RoboDK station: LEGOS_RDK.rdk

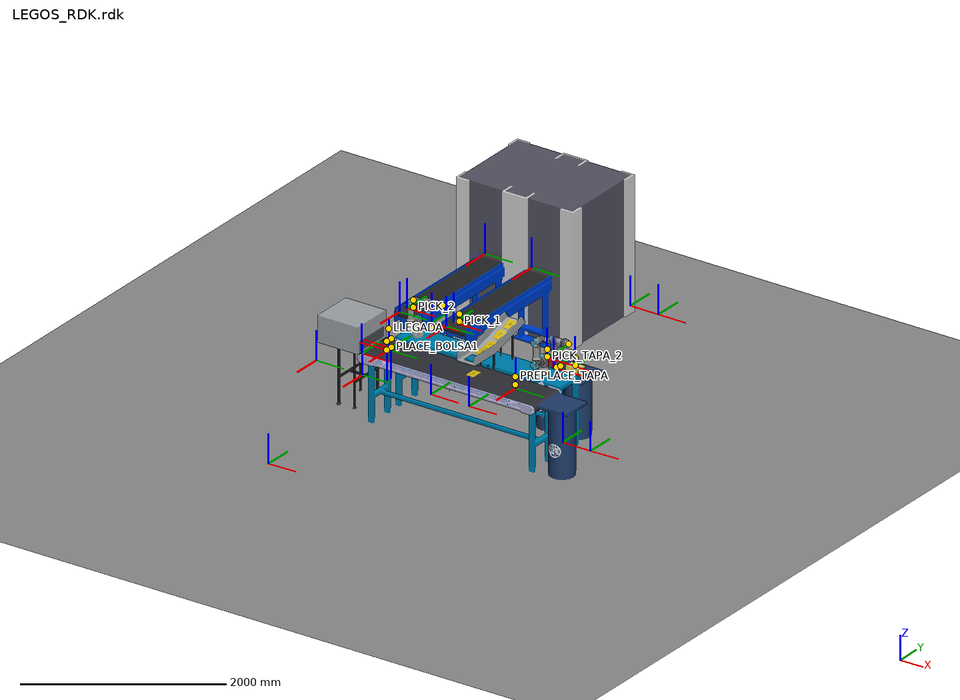
[picture v0: the station drawn from its stored meshes, robots at their saved joint values, targets as dots, program paths as lines]
Station LEGOS_RDK (saved by RoboDK 5.9.4). Poses are relative to the parent item; angles as X-Y-Z fixed-axis rotations.
Station parameters (name, value as stored): SenyalSensor_C, 0, SenyalSensor_T, 0, BOLSA2_PICK, 1, BOLSA1_PICK, 1, Continuar1, 1, PRIMERA_RUN, 1, SenyalSensor_I, 0, TOTAL_PEDIDO_1, 0, TOTAL_PEDIDO_2, 0, ACTIVO, 1, PP_BOLSA_2, 0, INS_BOLSA_2, 0, TAPA_BOLSA_2, 0, Conti_T, 1, lim_ins, 0, lim_tapa, 0, PARAR_ESTACION, 1, CICLOS_HASTA_PARAR, 0, PP_LOCAL, 0, IO_0, 0, Cinta_Terminada, 0, Conti_I, 1, MQTT_ESTACION_ENCENDIDA, 0, PARADA_EMERGENCIA, 0, INITIAL_P1, 0, CONTADOR_C, 2, CONTADOR_T, 2, lim_bolsa, 0, TOTAL_PEDIDO_2_INICIAL, 2, CONTADOR_I, 2, PEDIDO_1_INICIAL, 2, PEDIDO_2_INICIAL, 0, LIMITE_TAPAS, 0, LIMITE_INSTRU, 0, LIMITE_BOLSAS, 0, R1_LIBRE, 1, R2_LIBRE, 1, INSTRU_LIBRE, 1, PRODUCIR_CAJAS, 0, NUMERO_PEDIDO, PED_1779911272, STOCK_VERIFICADO, 1, ES_REANUDACION, 0, CONTADOR_CREADAS, 2, MAPA_CAJA_001, CAJA_001, MAPA_CAJA_002, CAJA_002, MAPA_CAJA_003, CAJA2_003, NOMBRE_C_001, CAJA_001, NOMBRE_C_002, CAJA_002, NOMBRE_T_001, instru_2, NOMBRE_T_002, instru_2, NOMBRE_T_003, instru_2, NOMBRE_C_003, CAJA2_003, NOMBRE_C_004, CAJA_004, MAPA_CAJA_004, CAJA_004, NOMBRE_C_005, CAJA_005, MAPA_CAJA_005, CAJA_005, NOMBRE_C_006, CAJA_005, MAPA_CAJA_006, CAJA_006, NOMBRE_C_007, CAJA_007, NOMBRE_T_004, instru_2, MAPA_CAJA_007, CAJA_007, NOMBRE_C_008, CAJA_008, NOMBRE_T_005, instru_2, MAPA_CAJA_008, CAJA_008, NOMBRE_C_009, CAJA_008, NOMBRE_T_006, instru_2, MAPA_CAJA_009, CAJA_009, NOMBRE_C_010, CAJA_010, NOMBRE_T_007, instru_2, MAPA_CAJA_010, CAJA_010, NOMBRE_T_008, instru_2, NOMBRE_T_009, instru_2, NOMBRE_T_010, instru_2, NOMBRE_CAJA_EN_T
  - frame ROBOT1 at (240, 410, 60) mm
    - frame Frame PEDESTAL (OBJETO 1) at (280, 230, -915) mm
      - frame COGIDA_1 at (-110, -105, 915) mm
        - target PICK_1 (Cartesian target) at (46.65, 33, 11.24) mm, rotated rx 180 ry 0 rz 0 deg; joints [76.028, -114.59, -95.798, -59.613, 90, -13.972] of r_UR3e_(COGIDA)
        - target PREPICK_1 (Cartesian target) at (46.65, 33, 90) mm, rotated rx 180 ry 0 rz 0 deg; joints [76.028, -108.102, -82.469, -79.429, 90, -13.972] of r_UR3e_(COGIDA)
    - frame Frame PEDESTAL (OBJETO 2) at (-170, 230, -915) mm
      - frame COGIDA_2 at (-210, -105, 915) mm
        - target PICK_2 (Cartesian target) at (46.65, 33, 11.24) mm, rotated rx 180 ry 0 rz 0 deg; joints [76.028, -114.59, -95.798, -59.613, 90, -13.972] of r_UR3e_(COGIDA)
        - target PREPICK_2 (Cartesian target) at (46.65, 33, 90) mm, rotated rx 180 ry 0 rz 0 deg; joints [76.028, -108.102, -82.469, -79.429, 90, -13.972] of r_UR3e_(COGIDA)
    - frame CircuitConveyor Base at (80, 125, -65) mm, rotated rx 0 ry 0 rz -90 deg
      - robot CircuitConveyorDoor: 1 axes
          modified DH rows (alpha deg, a mm, theta deg, d mm): 0, 0, 0, 0 linear
          joint limits [0] to [80]; home [0]; saved at [0]
      - frame CircuitConveyorRef_Init at (-1430, 10, 60) mm
        - object BOLSA 1 at (-120, 40, 0) mm, rotated rx 0 ry 0 rz -90 deg, size 93 x 60 x 20.1 mm, geometry from tinker.obj
      - robot CircuitConveyor: 1 axes
          modified DH rows (alpha deg, a mm, theta deg, d mm): 0, 0, 0, 0 linear
          base shift (0, 0, 0) mm, rotated rx 0 ry 90 rz 0 deg
          joint limits [-200000] to [200000]; home [0]; saved at [1430]
        - frame CircuitConveyorRef at (0, 10, 50) mm
          - object BOLSA 1 at (-1550, 40, 10) mm, rotated rx 0 ry 0 rz -90 deg, size 93 x 60 x 20.1 mm, geometry from tinker.obj
    - frame CircuitConveyor Base(2) at (-470, 125, -65) mm, rotated rx 0 ry 0 rz -90 deg
      - robot CircuitConveyorDoor(2): 1 axes
          modified DH rows (alpha deg, a mm, theta deg, d mm): 0, 0, 0, 0 linear
          joint limits [0] to [80]; home [0]; saved at [0]
      - frame CircuitConveyorRef_Init(2) at (-1430, 10, 60) mm
        - object BOLSA 2 at (-120, 40, 0) mm, rotated rx 0 ry 0 rz -90 deg, size 93 x 60 x 20.1 mm, geometry from tinker.obj
      - robot CircuitConveyor(2): 1 axes
          modified DH rows (alpha deg, a mm, theta deg, d mm): 0, 0, 0, 0 linear
          base shift (0, 0, 0) mm, rotated rx 0 ry 90 rz 0 deg
          joint limits [-200000] to [200000]; home [0]; saved at [1430]
        - frame CircuitConveyorRef(2) at (0, 10, 50) mm
          - object BOLSA 2 at (-1550, 40, 10) mm, rotated rx 0 ry 0 rz -90 deg, size 93 x 60 x 20.1 mm, geometry from tinker.obj
  - frame ROBOT 2 at (1680, 410, -20) mm
    - frame Frame PEDESTAL (PACK 2) at (-50, 230, -915) mm
      - object Pedestal H36in (Type 1) at (-110, -60, -69) mm, size 400 x 400 x 914.4 mm, geometry from Pedestal-H36in-Type-1.sld
      - object dispensa_tapas at (-122, -131, 835) mm, size 162 x 117 x 81 mm, geometry from tinker.obj
      - frame COGIDA_TAPA_2 at (-110, -105, 922) mm
        - target PICK_TAPA_2 (Cartesian target) at (0, 0, 11.24) mm, rotated rx 180 ry 0 rz 0 deg; joints [76.028, -114.59, -95.798, -59.613, 90, -13.972] of r_UR3e_(COGIDA)
        - target PREPICK_TAPA_2 (Cartesian target) at (0, 0, 90) mm, rotated rx 180 ry 0 rz 0 deg; joints [76.028, -108.102, -82.469, -79.429, 90, -13.972] of r_UR3e_(COGIDA)
        - frame FrameInitTapa_2 at (0, 1410, 0) mm
          - object TAPA at (-72, -1477.5, -10) mm, rotated rx 0 ry 0 rz 90 deg, size 111 x 156 x 21 mm, geometry from tinker.obj
        - object TAPA at (-72, -67.5, -10) mm, rotated rx 0 ry 0 rz 90 deg, size 111 x 156 x 21 mm, geometry from tinker.obj
    - frame Frame PEDESTAL (PACK 1) at (280, 230, -915) mm
      - object Pedestal H36in (Type 1) at (-110, -60, -69) mm, size 400 x 400 x 914.4 mm, geometry from Pedestal-H36in-Type-1.sld
      - object dispensa_tapas at (-122, -131, 835) mm, size 162 x 117 x 81 mm, geometry from tinker.obj
      - frame COGIDA_TAPA at (-110, -105, 922) mm
        - target PICK_TAPA (Cartesian target) at (0, 0, 11.24) mm, rotated rx 180 ry 0 rz 0 deg; joints [76.028, -114.59, -95.798, -59.613, 90, -13.972] of r_UR3e_(COGIDA)
        - target PREPICK_TAPA (Cartesian target) at (0, 0, 90) mm, rotated rx 180 ry 0 rz 0 deg; joints [76.028, -108.102, -82.469, -79.429, 90, -13.972] of r_UR3e_(COGIDA)
        - frame FrameInitTapa at (0, 1410, 0) mm
          - object TAPA at (-72, -1477.5, -10) mm, rotated rx 0 ry 0 rz 90 deg, size 111 x 156 x 21 mm, geometry from tinker.obj
        - object TAPA at (-72, -67.5, -10) mm, rotated rx 0 ry 0 rz 90 deg, size 111 x 156 x 21 mm, geometry from tinker.obj
  - frame FrameCintaP at (0, -440, 0) mm
    - robot CINTA_PRINCIPAL: 1 axes
        modified DH rows (alpha deg, a mm, theta deg, d mm): 0, 0, 0, 0 linear
        base shift (0, 0, 0) mm, rotated rx 0 ry 90 rz 0 deg
        joint limits [-500000] to [500000]; home [0]; saved at [0]
      - frame FrameCAJA at (170, 220, 0) mm, rotated rx 0 ry 0 rz -90 deg
    - object MesaCinta at (1040, 170, -770) mm, rotated rx 0 ry 0 rz -90 deg, size 320 x 2000 x 740 mm, geometry from tinker.obj
    - object Fotocelula_T at (1688, 448, 0) mm, rotated rx 90 ry 0 rz -90 deg, size 683.3 x 45.2 x 12.5 mm, geometry from SICK-WL4S-Laser-Sensor.sld
    - object Fotocelula_C at (188, 448, 0) mm, rotated rx 90 ry 0 rz -90 deg, size 683.3 x 45.2 x 12.5 mm, geometry from SICK-WL4S-Laser-Sensor.sld
    - object Fotocelula_I at (1188, 448, 0) mm, rotated rx 90 ry 0 rz -90 deg, size 683.3 x 45.2 x 12.5 mm, geometry from SICK-WL4S-Laser-Sensor.sld
    - frame COGIDA CINTA at (170, 220, 0) mm, rotated rx 0 ry 0 rz -90 deg
      - target LLEGADA (Cartesian target) at (0.04, 0.12, 230.39) mm, rotated rx -180 ry 0 rz -90 deg; joints [-75.94, -132.382, -21.795, -115.824, 90, 14.06] of r_UR3e_(COGIDA)
      - frame DEJAR_BOLSA1 at (-35, 2, 5) mm, rotated rx -180 ry 0 rz -90 deg
        - target PREPLACE_BOLSA1 (Cartesian target) at (0, 0, -100) mm; joints [-74.482, -118.64, -79.498, -71.862, 90, -344.482] of r_UR3e_(COGIDA)
        - target PLACE_BOLSA1 (Cartesian target) at (0, 0, -8) mm; joints [-74.482, -129.029, -89.848, -51.123, 90, -344.482] of r_UR3e_(COGIDA)
      - frame DEJAR_BOLSA2 at (35, 2, 5) mm, rotated rx -180 ry 0 rz -90 deg
        - target PREPLACE_BOLSA2 (Cartesian target) at (0, 0, -100) mm; joints [-74.482, -118.64, -79.498, -71.862, 90, -344.482] of r_UR3e_(COGIDA)
        - target PLACE_BOLSA2 (Cartesian target) at (0, 0, -8) mm; joints [-74.482, -129.029, -89.848, -51.123, 90, -344.482] of r_UR3e_(COGIDA)
    - frame LLEGADA CINTA at (1670, 220, 0) mm, rotated rx 0 ry 0 rz -90 deg
      - target PREPLACE_TAPA (Cartesian target) at (0, 0, 130) mm, rotated rx 180 ry 0 rz 180 deg; joints [-73.448, -126.178, -60.342, -83.48, 90, 106.552] of r_UR3e_(TAPAS)
      - target PLACE_TAPA (Cartesian target) at (0, 0, 45) mm, rotated rx 180 ry 0 rz 180 deg; joints [-73.448, -132.236, -73.608, -64.156, 90, 106.552] of r_UR3e_(TAPAS)
    - frame Frame_Mec_Cai at (-312, -1127, -825) mm
      - robot Mecanismo_Caida: 1 axes
          modified DH rows (alpha deg, a mm, theta deg, d mm): 0, 0, 0, 0 linear
          base shift (0, 0, 0) mm, rotated rx 0 ry 0 rz 90 deg
          joint limits [-163] to [0]; home [0]; saved at [-163]
    - frame Frame_dis_ins at (1170, 220, 0) mm, rotated rx 0 ry 0 rz -90 deg
      - object Dispensa_instru at (-180, 320, -270) mm, rotated rx 0 ry 0 rz 90 deg, size 216 x 857.7 x 462.8 mm, geometry from tinker.obj
      - object instru2 at (-20, -15, 180) mm, size 126 x 90 x 9.1 mm, geometry from tinker.obj
      - object Square at (0, 0, -10) mm, size 75 x 75 x 0 mm, geometry from Square.sld
    - frame FrameInitInstru at (0, 1410, 0) mm
      - object instru at (1155, -1170, 20) mm, rotated rx 0 ry 0 rz -90 deg, size 126 x 90 x 9.1 mm, geometry from tinker.obj
      - object instru_2 at (1155, -1170, 20) mm, rotated rx 0 ry 0 rz -90 deg, size 126 x 90 x 9.1 mm, geometry from tinker.obj
    - frame FrameInitCaja at (-330, 220, 0) mm, rotated rx 0 ry 0 rz -90 deg
      - object CAJA_REF at (-33, 18, 0) mm, size 105 x 150 x 39 mm, geometry from tinker.obj
      - object CAJA_REF_2 at (-33, 18, 0) mm, size 105 x 150 x 39 mm, geometry from tinker.obj
    - frame Frame_Disp_caj at (-312, 253, -825) mm
      - robot Dispensa_CAJAS: 1 axes
          modified DH rows (alpha deg, a mm, theta deg, d mm): 0, 0, 0, 0 linear
          base shift (0, 0, 0) mm, rotated rx 0 ry 0 rz 90 deg
          joint limits [0] to [120]; home [0]; saved at [0]
    - frame Frame_Caja_completa at (2330, 190, -850) mm, rotated rx 0 ry 0 rz 180 deg
      - object Pedestal H36in (Type 1) at (100, -20, -65) mm, size 400 x 400 x 914.4 mm, geometry from Pedestal-H36in-Type-1.sld
  - folder ROBOTS
    - frame UR3e_Base at (190, 240, -20) mm
      - robot r_UR3e_(COGIDA) (model UR3e): 6 axes, payload 3 kg, reach 500 mm, repeatability 0.03 mm, weight 11 kg
          modified DH rows (alpha deg, a mm, theta deg, d mm): 0, 0, 0, 151.9; 90, 0, 180, 0; 0, 243.55, 0, 0; 0, 213.2, 0, 131.05; -90, 0, 0, 85.35; 90, 0, 180, 92.1
          joint limits [-360, -360, -360, -360, -360, -360] to [360, 360, 360, 360, 360, 360]; home [0, -90, -90, 0, 90, 0]; saved at [0, -90, -90, 0, 90, 0]
        - tool VENTOSA-COG, TCP at (0, 0, 82.18) mm, size 70 x 70 x 80.4 mm
      - target HOME_R1 (Cartesian target) at (387.48, -131.05, 480.8) mm, rotated rx -90 ry 0 rz -90 deg; joints [37.926, -98.256, -58.971, -22.773, 52.074, 0] of r_UR3e_(COGIDA)
      - target SAFE_R1 (Cartesian target) at (298.55, -131.05, 221.17) mm, rotated rx -180 ry 0 rz -90 deg; joints [28.318, -100.412, -56.382, -113.206, 90, 28.318] of r_UR3e_(COGIDA)
      - target PUNTO_PASO_R1 (Cartesian target) at (319.11, -229.65, 250.13) mm, rotated rx -179.97 ry -0.01 rz -92.3 deg; joints [-16.27, -108.19, -60.7, -101.08, 90, -13.97] of r_UR3e_(COGIDA)
    - frame UR3e Base (2) at (1680, 240, -20) mm
      - robot r_UR3e_(TAPAS) (model UR3e): 6 axes, payload 3 kg, reach 500 mm, repeatability 0.03 mm, weight 11 kg
          modified DH rows (alpha deg, a mm, theta deg, d mm): 0, 0, 0, 151.9; 90, 0, 180, 0; 0, 243.55, 0, 0; 0, 213.2, 0, 131.05; -90, 0, 0, 85.35; 90, 0, 180, 92.1
          joint limits [-360, -360, -360, -360, -360, -360] to [360, 360, 360, 360, 360, 360]; home [0, -90, -90, 0, 90, 0]; saved at [0, -90, -90, 0, 90, 0]
        - tool VENTOSA-FIN, TCP at (0, 0, 82.18) mm, size 70 x 70 x 80.4 mm
      - target HOME_R2 (Cartesian target) at (387.48, -131.05, 480.8) mm, rotated rx -90 ry 0 rz -90 deg; joints [37.926, -98.256, -58.971, -22.773, 52.074, 0] of r_UR3e_(COGIDA)
      - target SAFE_R2 (Cartesian target) at (298.55, -131.05, 221.17) mm, rotated rx -180 ry 0 rz -90 deg; joints [28.318, -100.412, -56.382, -113.206, 90, 28.318] of r_UR3e_(COGIDA)
      - target PUNTO_PASO_R2 (Cartesian target) at (319.11, -229.65, 250.13) mm, rotated rx -179.97 ry -0.01 rz -92.3 deg; joints [-16.27, -108.19, -60.7, -101.08, 90, -13.97] of r_UR3e_(COGIDA)
      - target Target 4 (Cartesian target) at (298.55, -131.05, 221.17) mm, rotated rx -180 ry 0 rz -90 deg; joints [0, -90, -90, -90, 90, 0] of r_UR3e_(TAPAS)
  - folder OBJETOS SUELTOS
    - object Floor at (860, -90, -760) mm, size 9000 x 9000 x 0 mm, geometry from Floor.sld
    - frame Frame MESA_ROBOT at (940, 230, 0) mm
      - object Mesa_robots at (100, -40, -760) mm, rotated rx 0 ry 0 rz -90 deg, size 320 x 2000 x 740 mm, geometry from tinker.obj
  - folder PROGRAMAS PYTHON
    - Python program DetectaSensor (listed below)
    - Python program DISPENSAR_B1 (listed below)
    - Python program DISPENSAR_B2 (listed below)
    - Python program REPONER_TAPA (listed below)
    - Python program REPONER_TAPA_2 (listed below)
    - Python program PONER_INSTRU (listed below)
  - folder PROGRAMAS ROBOTS
    - Python program ROBOT1_BOLSA1 (listed below)
    - Python program ROBOT1_BOLSA2 (listed below)
    - Python program ROBOT2_TAPA1 (listed below)
    - Python program ROBOT2_TAPA2 (listed below)
  - Python program MAIN_PRODUCCION (listed below)
  - Python program MqttListener (listed below)
  - Python program BASE_DATOS (listed below)

--- Python program DetectaSensor ---
import time
from robodk import robolink
from robodk import robomath

"""
DetectaSensor.py — Script vigía de fotocélulas.
Corre como proceso independiente en paralelo con main_produccion.
Detecta colisiones entre las cajas del FrameCAJA y las tres fotocélulas
(C, I, T) y actualiza los params SenyalSensor_* en RoboDK.
Desde esta versión también escribe el NOMBRE de la caja detectada en
cada sensor ANTES de actualizar la señal, para que Base_datos pueda
identificar unívocamente qué caja física pasó por cada punto.
Se comunica con el resto de scripts ÚNICAMENTE vía RDK.setParam/getParam.
"""

RDK = robolink.Robolink()
RDK.COM.settimeout(10)

REFERENCE_FRAME = 'FrameCAJA'

frame = RDK.Item(REFERENCE_FRAME, robolink.ITEM_TYPE_FRAME)

fotocelulaC = RDK.Item('Fotocelula_C')
fotocelulaT = RDK.Item('Fotocelula_T')
fotocelulaI = RDK.Item('Fotocelula_I')

estado_detectadoC = -1
estado_detectadoT = -1
estado_detectadoI = -1

if not frame.Valid():
    raise Exception(f'El frame "{REFERENCE_FRAME}" no es válido o no existe.')

if not fotocelulaC.Valid() or not fotocelulaT.Valid() or not fotocelulaI.Valid():
    raise Exception('Alguna fotocélula no es válida (revisa los nombres de los ítems).')

while int(RDK.getParam('PARAR_ESTACION')) and int(RDK.getParam('PARADA_EMERGENCIA')) == 0:
    detectadoC = 0
    detectadoT = 0
    detectadoI = 0

    tipo_caja_C = '0'
    tipo_caja_T = '0'
    tipo_caja_I = '0'

    # Nombres de las cajas que están en cada sensor en esta iteración
    nombre_en_C = ''
    nombre_en_T = ''

    for item in frame.Childs():

        try:
            if not item.Valid() or item.Type() != robolink.ITEM_TYPE_OBJECT:
                continue

            nombre_caja = item.Name()
            nombre_upper = nombre_caja.upper()

            #  colisiones y guardamos la caja
            if fotocelulaC.Valid() and fotocelulaC.Collision(item):
                detectadoC  = 1
                nombre_en_C = nombre_caja
                if 'CAJA2' in nombre_upper:
                    tipo_caja_C = '1'

            if fotocelulaT.Valid() and fotocelulaT.Collision(item):
                detectadoT  = 1
                nombre_en_T = nombre_caja
                if 'CAJA2' in nombre_upper:
                    tipo_caja_T = '1'

            if fotocelulaI.Valid() and fotocelulaI.Collision(item):
                detectadoI = 1
                if 'CAJA2' in nombre_upper:
                    tipo_caja_I = '1'

        except Exception:
            continue

    # Escribir DATOS antes que SEÑALES
    RDK.setParam('PP_BOLSA_2',    tipo_caja_C)
    RDK.setParam('TAPA_BOLSA_2',  tipo_caja_T)
    RDK.setParam('INS_BOLSA_2',   tipo_caja_I)

    # Nombres de caja en sensor — Base_datos los lee para mapear
    RDK.setParam('NOMBRE_CAJA_EN_C', nombre_en_C)
    RDK.setParam('NOMBRE_CAJA_EN_T', nombre_en_T)

    # actualizamos los sensores si cambian
    if estado_detectadoC != detectadoC:
        RDK.setParam('SenyalSensor_C', str(detectadoC))
        estado_detectadoC = detectadoC

    if estado_detectadoT != detectadoT:
        RDK.setParam('SenyalSensor_T', str(detectadoT))
        estado_detectadoT = detectadoT

    if estado_detectadoI != detectadoI:
        RDK.setParam('SenyalSensor_I', str(detectadoI))
        estado_detectadoI = detectadoI

    time.sleep(0.1)

--- Python program DISPENSAR_B1 ---
from robodk import robolink
RDKCIRCUIT = robolink.Robolink()

"""
Stack Tecnológico: Python, RoboDK API (robolink).
Descripción: Script de ejecución lineal. Gestiona la clonación y dispensado
visual del objeto 'BOLSA 1' en la estación de suministro. Abre la compuerta,
avanza la cinta secundaria y la vuelve a cerrar.
"""

#----- Constante -----
NEW_REF_OBJECT_NAME = 'BOLSA 1'
NEW_OBJECT_NAME = 'BOLSAAA'
REFERENCE_FRAME = 'CircuitConveyorRef'
REFERENCE_FRAME_REF = 'CircuitConveyorRef_Init'
MECHANISM_NAME = 'CircuitConveyor'
MECHANISM_NAME_DOOR = 'CircuitConveyorDoor'

PART_TRAVEL_MM = 1430
DOOR_TRAVEL_MM = 56
N_DOOR_TRAVEL_MM = -56

mechanism = RDKCIRCUIT.Item(MECHANISM_NAME,itemtype=robolink.ITEM_TYPE_ROBOT)
door = RDKCIRCUIT.Item(MECHANISM_NAME_DOOR,itemtype=robolink.ITEM_TYPE_ROBOT)

#------- Programa ------
frame = RDKCIRCUIT.Item(REFERENCE_FRAME, robolink.ITEM_TYPE_FRAME)
frame_ref = RDKCIRCUIT.Item(REFERENCE_FRAME_REF, robolink.ITEM_TYPE_FRAME)
ref_obj = RDKCIRCUIT.Item(NEW_REF_OBJECT_NAME, robolink.ITEM_TYPE_OBJECT)


if mechanism.Valid():
    mechanism.setJoints([0])

if frame.Valid():
    for item in frame.Childs():
        if item.Type() == robolink.ITEM_TYPE_OBJECT:
            item.Delete()

RDKCIRCUIT.Render(False)

for item in frame_ref.Childs():
    if frame.Valid() and  ref_obj.Valid():
        item.Copy()
        new_obj = RDKCIRCUIT.Paste()
        new_obj.setVisible(False)
        new_obj.setParent(frame_ref)
        RDKCIRCUIT.Update()
        new_obj.setParentStatic(frame)
        new_obj.setVisible(True)

RDKCIRCUIT.Render(True)

if door.Valid():
    door.setJoints([0])

if door.Valid():
    door.MoveJ(door.Joints() + DOOR_TRAVEL_MM)

if mechanism.Valid():
    mechanism.MoveJ(mechanism.Joints() + PART_TRAVEL_MM)

if door.Valid():
    door.MoveJ(door.Joints() + N_DOOR_TRAVEL_MM)

RDKCIRCUIT.setParam('BOLSA1_PICK', '1')

--- Python program DISPENSAR_B2 ---
from robodk import robolink
RDKCIRCUIT = robolink.Robolink()

"""
Stack Tecnológico: Python 3, RoboDK API (robolink).
Descripción: Script de ejecución lineal. Gestiona la clonación y dispensado
visual del objeto 'BOLSA 2' en la estación de suministro, operando la
compuerta y la cinta secundaria asociada.
"""

#----- Constante -----
NEW_REF_OBJECT_NAME = 'BOLSA 2'
NEW_OBJECT_NAME = 'BOLSAAA'
REFERENCE_FRAME = 'CircuitConveyorRef(2)'
REFERENCE_FRAME_REF = 'CircuitConveyorRef_Init(2)'
MECHANISM_NAME = 'CircuitConveyor(2)'
MECHANISM_NAME_DOOR = 'CircuitConveyorDoor(2)'

PART_TRAVEL_MM = 1430
DOOR_TRAVEL_MM = 56
N_DOOR_TRAVEL_MM = -56

mechanism = RDKCIRCUIT.Item(MECHANISM_NAME,itemtype=robolink.ITEM_TYPE_ROBOT)
door = RDKCIRCUIT.Item(MECHANISM_NAME_DOOR,itemtype=robolink.ITEM_TYPE_ROBOT)

#------- Programa ------
frame = RDKCIRCUIT.Item(REFERENCE_FRAME, robolink.ITEM_TYPE_FRAME)
frame_ref = RDKCIRCUIT.Item(REFERENCE_FRAME_REF, robolink.ITEM_TYPE_FRAME)
ref_obj = RDKCIRCUIT.Item(NEW_REF_OBJECT_NAME, robolink.ITEM_TYPE_OBJECT)


if mechanism.Valid():
    mechanism.setJoints([0])

if frame.Valid():
    for item in frame.Childs():
        if item.Type() == robolink.ITEM_TYPE_OBJECT:
            item.Delete()

RDKCIRCUIT.Render(False)

for item in frame_ref.Childs():
    if frame.Valid() and  ref_obj.Valid():
        item.Copy()
        new_obj = RDKCIRCUIT.Paste()
        new_obj.setVisible(False)
        new_obj.setParent(frame_ref)
        RDKCIRCUIT.Update()
        new_obj.setParentStatic(frame)
        new_obj.setVisible(True)

RDKCIRCUIT.Render(True)

if door.Valid():
    door.setJoints([0])

if door.Valid():
    door.MoveJ(door.Joints() + DOOR_TRAVEL_MM)

if mechanism.Valid():
    mechanism.MoveJ(mechanism.Joints() + PART_TRAVEL_MM)

if door.Valid():
    door.MoveJ(door.Joints() + N_DOOR_TRAVEL_MM)

RDKCIRCUIT.setParam('BOLSA2_PICK', '1')

--- Python program REPONER_TAPA ---
from robodk import robolink
from robodk import robomath
RDKCIRCUIT = robolink.Robolink()

"""
Stack Tecnológico: Python, RoboDK API (robolink, robomath).
Descripción: Script de ejecución lineal. Se encarga de regenerar (clonar)
visualmente el modelo 3D de la 'TAPA' de Tipo 1 en el pedestal de recogida
una vez que el robot se ha llevado la anterior.
"""

#----- Constante -----
NEW_REF_OBJECT_NAME = 'TAPA'
NEW_OBJECT_NAME = 'TAPA_C'
REFERENCE_FRAME = 'COGIDA_TAPA'
REFERENCE_FRAME_REF = 'FrameInitTapa'

#------- Programa ------
frame = RDKCIRCUIT.Item(REFERENCE_FRAME, robolink.ITEM_TYPE_FRAME)
frame_ref = RDKCIRCUIT.Item(REFERENCE_FRAME_REF, robolink.ITEM_TYPE_FRAME)
ref_obj = RDKCIRCUIT.Item(NEW_REF_OBJECT_NAME, robolink.ITEM_TYPE_OBJECT)

if frame.Valid():
    for item in frame.Childs():
        if item.Type() == robolink.ITEM_TYPE_OBJECT:
            item.Delete()


RDKCIRCUIT.Render(False)

for item in frame_ref.Childs():
    if frame.Valid() and  ref_obj.Valid():
        item.Copy()
        new_obj = RDKCIRCUIT.Paste()
        new_obj.setVisible(False)
        new_obj.setParent(frame_ref)
        RDKCIRCUIT.Update()
        new_obj.setParentStatic(frame)
        new_obj.setVisible(True)

RDKCIRCUIT.Render(True)

--- Python program REPONER_TAPA_2 ---
from robodk import robolink
from robodk import robomath
RDKCIRCUIT = robolink.Robolink()

"""
Stack Tecnológico: Python 3, RoboDK API (robolink, robomath).
Descripción: Script de ejecución lineal. Regenera (clona) visualmente el
modelo 3D de la 'TAPA' de Tipo 2 en su pedestal específico para garantizar
el flujo continuo de abastecimiento al robot.
"""

#----- Constante -----
NEW_REF_OBJECT_NAME = 'TAPA'
NEW_OBJECT_NAME = 'TAPA_C'
REFERENCE_FRAME = 'COGIDA_TAPA_2'
REFERENCE_FRAME_REF = 'FrameInitTapa_2'

#------- Programa ------
frame = RDKCIRCUIT.Item(REFERENCE_FRAME, robolink.ITEM_TYPE_FRAME)
frame_ref = RDKCIRCUIT.Item(REFERENCE_FRAME_REF, robolink.ITEM_TYPE_FRAME)
ref_obj = RDKCIRCUIT.Item(NEW_REF_OBJECT_NAME, robolink.ITEM_TYPE_OBJECT)

if frame.Valid():
    for item in frame.Childs():
        if item.Type() == robolink.ITEM_TYPE_OBJECT:
            item.Delete()


RDKCIRCUIT.Render(False)

for item in frame_ref.Childs():
    if frame.Valid() and  ref_obj.Valid():
        item.Copy()
        new_obj = RDKCIRCUIT.Paste()
        new_obj.setVisible(False)
        new_obj.setParent(frame_ref)
        RDKCIRCUIT.Update()
        new_obj.setParentStatic(frame)
        new_obj.setVisible(True)

RDKCIRCUIT.Render(True)

--- Python program PONER_INSTRU ---
from robodk import robolink
from robodk import robomath
RDKCIRCUIT = robolink.Robolink()

"""
Stack Tecnológico: Python, RoboDK API (robolink, robomath).
Descripción: Script de ejecución lineal. Simula la inserción automática
de las instrucciones de montaje en el interior de las cajas. Mueve el
mecanismo de caída y clona visualmente el folleto en el frame destino.
"""

#----- Constante -----
NEW_REF_OBJECT_NAME = 'instru'
NEW_REF_OBJECT_NAME_2 = 'instru_2'
NEW_OBJECT_NAME = 'instru_c'
REFERENCE_FRAME = 'FrameCAJA'
REFERENCE_FRAME_REF = 'FrameInitInstru'

PART_TRAVEL_MM = -163
MECHANISM_NAME = 'Mecanismo_Caida'

#------- Programa ------
frame = RDKCIRCUIT.Item(REFERENCE_FRAME, robolink.ITEM_TYPE_FRAME)
frame_ref = RDKCIRCUIT.Item(REFERENCE_FRAME_REF, robolink.ITEM_TYPE_FRAME)
ref_obj = RDKCIRCUIT.Item(NEW_REF_OBJECT_NAME, robolink.ITEM_TYPE_OBJECT)
ref_obj_2 = RDKCIRCUIT.Item(NEW_REF_OBJECT_NAME_2, robolink.ITEM_TYPE_OBJECT)

mechanism = RDKCIRCUIT.Item(MECHANISM_NAME, robolink.ITEM_TYPE_ROBOT)

lim = int(RDKCIRCUIT.getParam('LIMITE_INSTRU'))


if lim != 0:

    #INCIAR CAIDA
    if mechanism.Valid():
        mechanism.setJoints([0])
        mechanism.setVisible(True)
        mechanism.MoveJ(mechanism.Joints() + PART_TRAVEL_MM)


    RDKCIRCUIT.Render(False)


    for item in frame_ref.Childs():
        if frame.Valid() and ref_obj.Valid():
            item.Copy()
            new_obj = RDKCIRCUIT.Paste()
            new_obj.setVisible(False)
            new_obj.setParent(frame_ref)
            RDKCIRCUIT.Update()
            new_obj.setParentStatic(frame)
            new_obj.setVisible(True)
            mechanism.setVisible(False)


    RDKCIRCUIT.Render(True)

    RDKCIRCUIT.setParam('INSTRU_LIBRE', '1')

--- Python program ROBOT1_BOLSA1 ---
import time

from robodk import robolink    # RoboDK API
from robodk import robomath    # Robot toolbox
from robolink import *
RDK = robolink.Robolink()

"""
Stack Tecnológico: Python 3, RoboDK API.
Descripción: Script cinemático del Robot 1 (UR3e de Cogida).
Contiene las rutinas de movimiento exactas (MoveJ, MoveL) para
coger bolsas de las estaciones secundarias y dejarlas en las cajas.
"""

robot = RDK.Item('r_UR3e_(COGIDA)', robolink.ITEM_TYPE_ROBOT)
tool = RDK.Item('VENTOSA-COG', robolink.ITEM_TYPE_TOOL)

#FRAMES
frame_robot = RDK.Item('UR3e_Base', robolink.ITEM_TYPE_FRAME)
frame_zt_rb1 = RDK.Item('ROBOT1', robolink.ITEM_TYPE_FRAME)
frame_at_1_rb1 = RDK.Item('Frame PEDESTAL (OBJETO 1)', robolink.ITEM_TYPE_FRAME)
frame_at_1_rb1_cog = RDK.Item('COGIDA_1', robolink.ITEM_TYPE_FRAME)

frame_cinta = RDK.Item('FrameCintaP', robolink.ITEM_TYPE_FRAME)
frame_cinta_aprox = RDK.Item('COGIDA CINTA', robolink.ITEM_TYPE_FRAME)
frame_cinta_b1 = RDK.Item('DEJAR_BOLSA1', robolink.ITEM_TYPE_FRAME)
frame_cinta_b2 = RDK.Item('DEJAR_BOLSA2', robolink.ITEM_TYPE_FRAME)


#TARGETS
home = RDK.Item('HOME_R1', robolink.ITEM_TYPE_TARGET)
safe = RDK.Item('SAFE_R1', robolink.ITEM_TYPE_TARGET)
punto_paso = RDK.Item('PUNTO_PASO_R1', robolink.ITEM_TYPE_TARGET)

pick_bolsa_1 = RDK.Item('PICK_1', robolink.ITEM_TYPE_TARGET)
prepick_bolsa_1 = RDK.Item('PREPICK_1', robolink.ITEM_TYPE_TARGET)

llegada_caja = RDK.Item('LLEGADA', robolink.ITEM_TYPE_TARGET)
llegada_caja_b1_preplace = RDK.Item('PREPLACE_BOLSA1', robolink.ITEM_TYPE_TARGET)
llegada_caja_b1_place = RDK.Item('PLACE_BOLSA1', robolink.ITEM_TYPE_TARGET)
llegada_caja_b2_preplace = RDK.Item('PREPLACE_BOLSA2', robolink.ITEM_TYPE_TARGET)
llegada_caja_b2_place = RDK.Item('PLACE_BOLSA2', robolink.ITEM_TYPE_TARGET)

#VARIABLES


# Asignar la herramienta al robot
robot.setTool(tool)

def Pick_b1(r):
    """
    Realiza la maniobra de aproximación, cogida y retroceso de una Bolsa Tipo 1.
    Espera a que el dispensador genere la bolsa antes de iniciar el movimiento.
    Adjunta el objeto 3D a la herramienta (ventosa).

    r (Item): El objeto robot de RoboDK que realizará el movimiento.
    """
    while int(RDK.getParam('BOLSA1_PICK')) != 1 and int(RDK.getParam('PARADA_EMERGENCIA')) == 0:
        time.sleep(0.1)

    if int(RDK.getParam('PARADA_EMERGENCIA')) == 1:
        return

    velocidad_lineal = 400
    robot.setSpeed(velocidad_lineal)

    r.setPoseFrame(frame_at_1_rb1_cog)
    r.MoveJ(prepick_bolsa_1)

    velocidad_lineal = 50
    r.setSpeed(velocidad_lineal)

    r.MoveL(pick_bolsa_1)

    #ADJUNTAR OBJETO A VENTOSA
    tool.AttachClosest()

    RDK.setParam('BOLSA1_PICK', '0')
    r.Pause(1000)
    r.MoveL(prepick_bolsa_1)

    velocidad_lineal = 400
    robot.setSpeed(velocidad_lineal)


def Place_bolsa1_tipo1(r):
    """
    Realiza la maniobra de posicionamiento y liberación (Place) de la Bolsa Tipo 1
    en el compartimento 2 de la caja (por requisitos del Tipo 1).
    Detacha la bolsa de la ventosa al Frame de la caja.
    """

    RDK.RunProgram('DISPENSAR_B1', False)

    if int(RDK.getParam('PARADA_EMERGENCIA')) == 1:
        return

    r.setPoseFrame(frame_cinta_aprox)
    r.MoveJ(llegada_caja)

    r.setPoseFrame(frame_cinta_b2)
    r.MoveL(llegada_caja_b2_preplace)

    velocidad_lineal = 50
    r.setSpeed(velocidad_lineal)

    r.MoveL(llegada_caja_b2_place)

    #LIBERAR BOLSA
    frame_destino = RDK.Item('FrameCAJA', ITEM_TYPE_FRAME)
    tool.DetachAll(frame_destino)

    r.Pause(1000)
    r.MoveL(llegada_caja_b2_preplace)

    velocidad_lineal = 400
    r.setSpeed(velocidad_lineal)


def Place_bolsa2_tipo1(r):
    """
    Realiza la maniobra de posicionamiento y liberación (Place) de la segunda Bolsa
    en el compartimento 1 de la caja.
    """

    RDK.RunProgram('DISPENSAR_B1', False)

    if int(RDK.getParam('PARADA_EMERGENCIA')) == 1:
        return

    r.setPoseFrame(frame_cinta_aprox)
    r.MoveJ(llegada_caja)

    r.setPoseFrame(frame_cinta_b1)
    r.MoveL(llegada_caja_b1_preplace)

    velocidad_lineal = 50
    r.setSpeed(velocidad_lineal)

    r.MoveL(llegada_caja_b1_place)

    #LIBERAR BOLSA
    frame_destino = RDK.Item('FrameCAJA', ITEM_TYPE_FRAME)
    tool.DetachAll(frame_destino)

    r.Pause(1000)
    r.MoveL(llegada_caja_b1_preplace)

    velocidad_lineal = 400
    r.setSpeed(velocidad_lineal)


def PickAndPlace_b_tipo1(r):
    """
    Rutina completa para empaquetar una Caja Tipo 1.
    Encadena secuencialmente los movimientos de Home -> Safe -> Pick -> Punto de Paso
    -> Place (repetido para las dos bolsas) y devuelve el control a la cinta.
    """
    if int(RDK.getParam('PARADA_EMERGENCIA')) == 1:
        return

    RDK.setParam('R1_LIBRE', '0')

    r.setPoseFrame(frame_robot)

    r.MoveJ(safe)

    Pick_b1(robot)

    r.setPoseFrame(frame_robot)
    r.MoveJ(punto_paso)

    Place_bolsa1_tipo1(robot)

    r.setPoseFrame(frame_robot)
    r.MoveJ(safe)

    Pick_b1(robot)

    r.setPoseFrame(frame_robot)
    r.MoveJ(punto_paso)

    Place_bolsa2_tipo1(robot)

    r.setPoseFrame(frame_robot)
    r.MoveJ(safe)

    RDK.setParam('R1_LIBRE', '1')


PickAndPlace_b_tipo1(robot)

--- Python program ROBOT1_BOLSA2 ---
import time

from robodk import robolink    # RoboDK API
from robodk import robomath    # Robot toolbox
from robolink import *
RDK = robolink.Robolink()

"""
========================================================
Stack Tecnológico: Python, RoboDK API.
Descripción: Script cinemático del Robot 1
Contiene las rutinas de movimiento exactas (MoveJ, MoveL) para
coger bolsas de las estaciones secundarias y dejarlas en las cajas.
========================================================
"""

robot = RDK.Item('r_UR3e_(COGIDA)', robolink.ITEM_TYPE_ROBOT)
tool = RDK.Item('VENTOSA-COG', robolink.ITEM_TYPE_TOOL)

#FRAMES
frame_robot = RDK.Item('UR3e_Base', robolink.ITEM_TYPE_FRAME) #Estan los targets basicos (home, safe, pp)
frame_zt_rb1 = RDK.Item('ROBOT1', robolink.ITEM_TYPE_FRAME)
frame_at_2_rb1 = RDK.Item('Frame PEDESTAL (OBJETO 2)', robolink.ITEM_TYPE_FRAME)
frame_at_2_rb1_cog = RDK.Item('COGIDA_2', robolink.ITEM_TYPE_FRAME)

frame_cinta = RDK.Item('FrameCintaP', robolink.ITEM_TYPE_FRAME)
frame_cinta_aprox = RDK.Item('COGIDA CINTA', robolink.ITEM_TYPE_FRAME)
frame_cinta_b1 = RDK.Item('DEJAR_BOLSA1', robolink.ITEM_TYPE_FRAME)
frame_cinta_b2 = RDK.Item('DEJAR_BOLSA2', robolink.ITEM_TYPE_FRAME)


#TARGETS
home = RDK.Item('HOME_R1', robolink.ITEM_TYPE_TARGET)
safe = RDK.Item('SAFE_R1', robolink.ITEM_TYPE_TARGET)
punto_paso = RDK.Item('PUNTO_PASO_R1', robolink.ITEM_TYPE_TARGET)

pick_bolsa_2 = RDK.Item('PICK_2', robolink.ITEM_TYPE_TARGET)
prepick_bolsa_2 = RDK.Item('PREPICK_2', robolink.ITEM_TYPE_TARGET)

llegada_caja = RDK.Item('LLEGADA', robolink.ITEM_TYPE_TARGET)
llegada_caja_b1_preplace = RDK.Item('PREPLACE_BOLSA1', robolink.ITEM_TYPE_TARGET)
llegada_caja_b1_place = RDK.Item('PLACE_BOLSA1', robolink.ITEM_TYPE_TARGET)
llegada_caja_b2_preplace = RDK.Item('PREPLACE_BOLSA2', robolink.ITEM_TYPE_TARGET)
llegada_caja_b2_place = RDK.Item('PLACE_BOLSA2', robolink.ITEM_TYPE_TARGET)

#VARIABLES


# Asignar la herramienta al robot
robot.setTool(tool)

def Pick_b2(r):
    """
    Realiza la maniobra de aproximación, cogida y retroceso de una Bolsa Tipo 2.
    Espera a que el dispensador genere la bolsa antes de iniciar el movimiento.
    Adjunta el objeto 3D a la herramienta (ventosa).

    r (Item): El objeto robot de RoboDK que realizará el movimiento.
    """
    while int(RDK.getParam('BOLSA2_PICK')) != 1 and int(RDK.getParam('PARADA_EMERGENCIA')) == 0:
        time.sleep(0.1)

    if int(RDK.getParam('PARADA_EMERGENCIA')) == 1:
        return

    velocidad_lineal = 400
    robot.setSpeed(velocidad_lineal)

    r.setPoseFrame(frame_at_2_rb1_cog)
    r.MoveJ(prepick_bolsa_2)

    velocidad_lineal = 50
    r.setSpeed(velocidad_lineal)

    r.MoveL(pick_bolsa_2)

    #ADJUNTAR OBJETO A VENTOSA
    tool.AttachClosest()

    RDK.setParam('BOLSA2_PICK', '0')
    r.Pause(1000)
    r.MoveL(prepick_bolsa_2)

    velocidad_lineal = 400
    robot.setSpeed(velocidad_lineal)


def Place_bolsa1_tipo2(r):
    """
    Realiza la maniobra de posicionamiento y liberación (Place) de la Bolsa Tipo 2
    en el compartimento 1 de la caja.
    Detacha la bolsa de la ventosa al Frame de la caja.
    """

    RDK.RunProgram('DISPENSAR_B2', False)

    if int(RDK.getParam('PARADA_EMERGENCIA')) == 1:
        return

    r.setPoseFrame(frame_cinta_aprox)
    r.MoveJ(llegada_caja)

    r.setPoseFrame(frame_cinta_b2)
    r.MoveL(llegada_caja_b2_preplace)

    velocidad_lineal = 50
    r.setSpeed(velocidad_lineal)

    r.MoveL(llegada_caja_b2_place)

    #LIBERAR BOLSA
    frame_destino = RDK.Item('FrameCAJA', ITEM_TYPE_FRAME)
    tool.DetachAll(frame_destino)

    r.Pause(1000)
    r.MoveL(llegada_caja_b2_preplace)

    velocidad_lineal = 400
    r.setSpeed(velocidad_lineal)


def Place_bolsa2_tipo2(r):
    """
    Realiza la maniobra de posicionamiento y liberación (Place) de la segunda Bolsa
    en el compartimento 2 de la caja.
    """

    RDK.RunProgram('DISPENSAR_B2', False)

    if int(RDK.getParam('PARADA_EMERGENCIA')) == 1:
        return

    r.setPoseFrame(frame_cinta_aprox)
    r.MoveJ(llegada_caja)

    r.setPoseFrame(frame_cinta_b1)
    r.MoveL(llegada_caja_b1_preplace)

    velocidad_lineal = 50
    r.setSpeed(velocidad_lineal)

    r.MoveL(llegada_caja_b1_place)

    #LIBERAR BOLSA
    frame_destino = RDK.Item('FrameCAJA', ITEM_TYPE_FRAME)
    tool.DetachAll(frame_destino)

    r.Pause(1000)
    r.MoveL(llegada_caja_b1_preplace)

    velocidad_lineal = 400
    r.setSpeed(velocidad_lineal)


def PickAndPlace_b_tipo2(r):
    """
    Rutina completa para empaquetar una Caja Tipo 2.
    Encadena secuencialmente los movimientos de Home -> Safe -> Pick -> Punto de Paso
    -> Place (repetido para las dos bolsas) y devuelve el control a la cinta.
    """
    if int(RDK.getParam('PARADA_EMERGENCIA')) == 1:
        return

    RDK.setParam('R1_LIBRE', '0')

    r.setPoseFrame(frame_robot)

    r.MoveJ(safe)

    Pick_b2(robot)

    r.setPoseFrame(frame_robot)
    r.MoveJ(punto_paso)

    Place_bolsa1_tipo2(robot)

    r.setPoseFrame(frame_robot)
    r.MoveJ(safe)

    Pick_b2(robot)

    r.setPoseFrame(frame_robot)
    r.MoveJ(punto_paso)

    Place_bolsa2_tipo2(robot)

    r.setPoseFrame(frame_robot)
    r.MoveJ(safe)

    RDK.setParam('R1_LIBRE', '1')


PickAndPlace_b_tipo2(robot)

--- Python program ROBOT2_TAPA1 ---
import time

from robodk import robolink    # RoboDK API
from robodk import robomath    # Robot toolbox
from robolink import *
RDK = robolink.Robolink()

"""
Stack Tecnológico: Python, RoboDK API (robolink, robomath).
Descripción: Script cinemático del Robot 2 (UR3e de Tapas).
Contiene las rutinas de movimiento exactas para recoger la Tapa Tipo 1
desde el pedestal y colocarla de forma precisa sobre la caja en la cinta.
"""

robot = RDK.Item('r_UR3e_(TAPAS)', robolink.ITEM_TYPE_ROBOT)
tool = RDK.Item('VENTOSA-FIN', robolink.ITEM_TYPE_TOOL)

#FRAMES
frame_robot = RDK.Item('UR3e Base (2)', robolink.ITEM_TYPE_FRAME) #Estan los targets basicos (home, safe, pp)
frame_zt_rb2 = RDK.Item('ROBOT2', robolink.ITEM_TYPE_FRAME)
frame_at_1_rb2 = RDK.Item('Frame PEDESTAL (PACK 1)', robolink.ITEM_TYPE_FRAME)
frame_at_2_rb1_cog = RDK.Item('COGIDA_TAPA', robolink.ITEM_TYPE_FRAME)

frame_cinta = RDK.Item('FrameCintaP', robolink.ITEM_TYPE_FRAME)
frame_cinta_aprox = RDK.Item('LLEGADA CINTA', robolink.ITEM_TYPE_FRAME)


#TARGETS
home = RDK.Item('HOME_R2', robolink.ITEM_TYPE_TARGET)
safe = RDK.Item('SAFE_R2', robolink.ITEM_TYPE_TARGET)
punto_paso = RDK.Item('PUNTO_PASO_R2', robolink.ITEM_TYPE_TARGET)

pick_tapa_2 = RDK.Item('PICK_TAPA', robolink.ITEM_TYPE_TARGET)
prepick_tapa_2 = RDK.Item('PREPICK_TAPA', robolink.ITEM_TYPE_TARGET)

tapa_preplace = RDK.Item('PREPLACE_TAPA', robolink.ITEM_TYPE_TARGET)
tapa_place = RDK.Item('PLACE_TAPA', robolink.ITEM_TYPE_TARGET)

#VARIABLES


# Asignar la herramienta al robot
robot.setTool(tool)

def Pick_tapa1(r):
    """
    Realiza la maniobra de aproximación, sujeción y retroceso de una Tapa Tipo 1.
    Adjunta el objeto 3D a la ventosa final, cambia el estado de la señal IO_0
    y ejecuta el script de reposición de tapas para preparar la siguiente.

    r (Item): El objeto robot de RoboDK que realizará el movimiento.
    """
    if int(RDK.getParam('PARADA_EMERGENCIA')) == 1:
        return

    velocidad_lineal = 400
    robot.setSpeed(velocidad_lineal)

    r.setPoseFrame(frame_at_2_rb1_cog)
    r.MoveJ(prepick_tapa_2)

    velocidad_lineal = 50
    r.setSpeed(velocidad_lineal)

    r.MoveL(pick_tapa_2)

    #ADJUNTAR OBJETO A VENTOSA
    tool.AttachClosest()

    r.Pause(1000)
    r.MoveL(prepick_tapa_2)

    velocidad_lineal = 400
    robot.setSpeed(velocidad_lineal)



def Place_tapa1(r):
    """
    Realiza la maniobra de posicionamiento y liberación (Place) de la Tapa Tipo 1
    sobre la caja en la cinta transportadora.
    Desvincula la tapa de la ventosa dejándola hija del Frame de la caja.
    """
    RDK.RunProgram('REPONER_TAPA', False)

    if int(RDK.getParam('PARADA_EMERGENCIA')) == 1:
        return

    r.setPoseFrame(frame_cinta_aprox)
    r.MoveJ(tapa_preplace)

    velocidad_lineal = 50
    r.setSpeed(velocidad_lineal)

    r.MoveL(tapa_place)

    #LIBERAR TAPA
    frame_destino = RDK.Item('FrameCAJA', ITEM_TYPE_FRAME)
    tool.DetachAll(frame_destino)

    r.Pause(1000)
    r.MoveL(tapa_preplace)

    velocidad_lineal = 400
    r.setSpeed(velocidad_lineal)


def PickAndPlace_tapa_tipo1(r):
    """
    Rutina completa para el sellado de una Caja Tipo 1.
    Detiene la señal de avance de cinta, encadena secuencialmente los movimientos
    (Safe -> Pick -> Punto de Paso -> Place -> Safe) y vuelve a permitir el avance de la cinta.
    """
    if int(RDK.getParam('PARADA_EMERGENCIA')) == 1:
        return

    RDK.setParam('R2_LIBRE', '0')

    r.setPoseFrame(frame_robot)

    r.MoveJ(safe)

    Pick_tapa1(robot)

    r.setPoseFrame(frame_robot)
    r.MoveJ(punto_paso)

    Place_tapa1(robot)

    r.setPoseFrame(frame_robot)
    r.MoveJ(safe)

    RDK.setParam('R2_LIBRE', '1')


PickAndPlace_tapa_tipo1(robot)

--- Python program ROBOT2_TAPA2 ---
import time

from robodk import robolink    # RoboDK API
from robodk import robomath    # Robot toolbox
from robolink import *
RDK = robolink.Robolink()

"""
Stack Tecnológico: Python 3.x, RoboDK API (robolink, robomath).
Descripción: Script cinemático del Robot 2 (UR3e de Tapas).
Contiene las rutinas de movimiento exactas para recoger la Tapa Tipo 2
desde su respectivo pedestal y colocarla sobre la caja correspondiente.
"""

robot = RDK.Item('r_UR3e_(TAPAS)', robolink.ITEM_TYPE_ROBOT)
tool = RDK.Item('VENTOSA-FIN', robolink.ITEM_TYPE_TOOL)

#FRAMES
frame_robot = RDK.Item('UR3e Base (2)', robolink.ITEM_TYPE_FRAME) #Estan los targets basicos (home, safe, pp)
frame_zt_rb2 = RDK.Item('ROBOT2', robolink.ITEM_TYPE_FRAME)
frame_at_2_rb2 = RDK.Item('Frame PEDESTAL (PACK 2)', robolink.ITEM_TYPE_FRAME)
frame_at_2_rb2_cog = RDK.Item('COGIDA_TAPA_2', robolink.ITEM_TYPE_FRAME)

frame_cinta = RDK.Item('FrameCintaP', robolink.ITEM_TYPE_FRAME)
frame_cinta_aprox = RDK.Item('LLEGADA CINTA', robolink.ITEM_TYPE_FRAME)


#TARGETS
home = RDK.Item('HOME_R2', robolink.ITEM_TYPE_TARGET)
safe = RDK.Item('SAFE_R2', robolink.ITEM_TYPE_TARGET)
punto_paso = RDK.Item('PUNTO_PASO_R2', robolink.ITEM_TYPE_TARGET)

pick_tapa_2 = RDK.Item('PICK_TAPA_2', robolink.ITEM_TYPE_TARGET)
prepick_tapa_2 = RDK.Item('PREPICK_TAPA_2', robolink.ITEM_TYPE_TARGET)

tapa_preplace = RDK.Item('PREPLACE_TAPA', robolink.ITEM_TYPE_TARGET)
tapa_place = RDK.Item('PLACE_TAPA', robolink.ITEM_TYPE_TARGET)

#VARIABLES


# Asignar la herramienta al robot
robot.setTool(tool)

def Pick_tapa2(r):
    """
    Realiza la maniobra de aproximación, sujeción y retroceso de una Tapa Tipo 2.
    Adjunta el objeto a la ventosa, pausa la simulación 1000ms para asegurar el agarre
    y repone una nueva Tapa Tipo 2 en el pedestal.

    r (Item): El objeto robot de RoboDK que realizará el movimiento.
    """
    if int(RDK.getParam('PARADA_EMERGENCIA')) == 1:
        return

    velocidad_lineal = 400
    r.setSpeed(velocidad_lineal)

    r.setPoseFrame(frame_at_2_rb2_cog)
    r.MoveJ(prepick_tapa_2)

    velocidad_lineal = 50
    r.setSpeed(velocidad_lineal)

    r.MoveL(pick_tapa_2)

    #ADJUNTAR OBJETO A VENTOSA
    tool.AttachClosest()

    r.Pause(1000)
    r.MoveL(prepick_tapa_2)

    velocidad_lineal = 400
    robot.setSpeed(velocidad_lineal)


def Place_tapa2(r):
    """
    Realiza la maniobra de posicionamiento y liberación (Place) de la Tapa Tipo 2
    sobre la caja en la cinta transportadora principal.
    """
    RDK.RunProgram('REPONER_TAPA_2', False)

    if int(RDK.getParam('PARADA_EMERGENCIA')) == 1:
        return

    r.setPoseFrame(frame_cinta_aprox)
    r.MoveJ(tapa_preplace)

    velocidad_lineal = 50
    r.setSpeed(velocidad_lineal)

    r.MoveL(tapa_place)

    #LIBERAR TAPA
    frame_destino = RDK.Item('FrameCAJA', ITEM_TYPE_FRAME)
    tool.DetachAll(frame_destino)

    r.Pause(1000)
    r.MoveL(tapa_preplace)

    velocidad_lineal = 400
    r.setSpeed(velocidad_lineal)


def PickAndPlace_tapa_tipo2(r):
    """
    Rutina completa para el sellado de una Caja Tipo 2.
    Bloquea el flujo de la estación, ejecuta las rutinas de Pick y Place
    utilizando puntos de paso seguros, y restaura la continuidad.
    """
    if int(RDK.getParam('PARADA_EMERGENCIA')) == 1:
        return

    RDK.setParam('R2_LIBRE', '0')

    r.setPoseFrame(frame_robot)

    r.MoveJ(safe)

    Pick_tapa2(robot)

    r.setPoseFrame(frame_robot)
    r.MoveJ(punto_paso)

    Place_tapa2(robot)

    r.setPoseFrame(frame_robot)
    r.MoveJ(safe)

    RDK.setParam('R2_LIBRE', '1')


PickAndPlace_tapa_tipo2(robot)

--- Python program MAIN_PRODUCCION ---
import time
from robodk import robolink
from robodk import robomath
from robolink import *
RDK = robolink.Robolink()

"""
Stack Tecnológico: Python, RoboDK API (robolink, robomath).
Descripción: Script principal (Main) que orquesta la estación.
Gestiona el inicio, los bucles de la cinta transportadora, las
llamadas a los robots y el control de paradas de emergencia.
"""

def Reset():
    """
    Limpia el entorno 3D antes de esperar un nuevo pedido:
    borra las cajas del frame 'FrameCAJA', reinicia la posición
    de la cinta y asegura que la señal MQTT de encendido esté a 0.
    Si venimos de una emergencia, NO borra las cajas para poder reanudar.
    """
    emergencia_activa = int(RDK.getParam('PARADA_EMERGENCIA') or '0') == 1

    RDK.setParam('MQTT_ESTACION_ENCENDIDA', '0')
    RDK.setParam('PARAR_ESTACION', '1')

    if emergencia_activa:
        # Si estamos en emergencia, salimos de la función sin borrar los objetos
        return

    REFERENCE_FRAME = 'FrameCAJA'
    frame = RDK.Item(REFERENCE_FRAME, robolink.ITEM_TYPE_FRAME)
    cinta = RDK.Item('CINTA_PRINCIPAL')

    if cinta.Valid():
        cinta.setJoints([0, 18, 0])

    # BORRAR LOS OBJETOS SITUADOS EN FRAME
    if frame.Valid():
        for item in frame.Childs():
            if item.Type() == robolink.ITEM_TYPE_OBJECT:
                item.Delete()

def init():
    """
    Inicializa todos los parámetros de RoboDK antes de arrancar un pedido.
    Calcula los límites de ciclos para cada sensor y devuelve los robots a posición HOME.
    Debe llamarse una única vez tras recibir la señal MQTT de inicio.
    """
    #Indicar que es el principio de un pedido (sin emergencia)
    es_reanudacion = int(RDK.getParam('ES_REANUDACION') or '0') == 1

    #Quitar la parada de emergenia para evitar confusion en otros pedidos
    RDK.setParam('PARADA_EMERGENCIA', '0')
    RDK.setParam('PRODUCIR_CAJAS', '1')

    #Resetear la verificacion de stock para el pedido actual
    RDK.setParam('STOCK_VERIFICADO', '0')

    if not es_reanudacion:
        # Guardar el total inicial de pedido 1 como referencia fija
        p1 = int(RDK.getParam('TOTAL_PEDIDO_1'))
        p2 = int(RDK.getParam('TOTAL_PEDIDO_2'))
        RDK.setParam('PEDIDO_1_INICIAL', str(p1))
        RDK.setParam('PEDIDO_2_INICIAL', str(p2))

        # Contadores de cajas que han llegado a cada sensor
        RDK.setParam('CONTADOR_C', '0')
        RDK.setParam('CONTADOR_T', '0')
        RDK.setParam('CONTADOR_I', '0')

        #Contador de cajas creadas para generar nombres distintos
        RDK.setParam('CONTADOR_CREADAS', '0')

        # Resetear la cuenta de cajas
        RDK.setParam('BOLSA1_PICK', '1')
        RDK.setParam('BOLSA2_PICK', '1')

        # INICIALIZAR VARIABLES PARA INDICAR QUE ES LA SEGUNDA CAJA POR MONTAR
        RDK.setParam('PP_BOLSA_2', '0')
        RDK.setParam('INS_BOLSA_2', '0')
        RDK.setParam('TAPA_BOLSA_2', '0')

        # LEYENDO PEDIDOS DE MQTT
        total_cajas = p1 + p2

        #Variables para indicar cuando acaban de moverse los robots
        #Se pone más para que el sistema y las variables se actualicen
        LIMITE_TAPAS = total_cajas + 4
        LIMITE_INSTRU = total_cajas + 3
        LIMITE_BOLSAS = total_cajas + 1
        RDK.setParam('LIMITE_TAPAS', str(LIMITE_TAPAS))
        RDK.setParam('LIMITE_INSTRU', str(LIMITE_INSTRU))
        RDK.setParam('LIMITE_BOLSAS', str(LIMITE_BOLSAS))

        stop = total_cajas + 12
        RDK.setParam('CICLOS_HASTA_PARAR', str(stop))
    else:
        # si se reanuda después de una emergencia conservar contadores y límites
        # Solo recalcular CICLOS_HASTA_PARAR con lo que queda
        p1 = int(RDK.getParam('TOTAL_PEDIDO_1'))
        p2 = int(RDK.getParam('TOTAL_PEDIDO_2'))

        restantes = p1 + p2 + 12
        RDK.setParam('CICLOS_HASTA_PARAR', str(restantes))

    # Variables de sincronización de cinta
    RDK.setParam('R1_LIBRE', '1')
    RDK.setParam('R2_LIBRE', '1')
    RDK.setParam('INSTRU_LIBRE', '1')

    #Devolver los robots a sus posiciones iniciales
    robot_1 = RDK.Item('r_UR3e_(COGIDA)', robolink.ITEM_TYPE_ROBOT)
    tool_1 = RDK.Item('VENTOSA-COG', robolink.ITEM_TYPE_TOOL)

    robot_2 = RDK.Item('r_UR3e_(TAPAS)', robolink.ITEM_TYPE_ROBOT)
    tool_2 = RDK.Item('VENTOSA-FIN', robolink.ITEM_TYPE_TOOL)

    #FRAMES
    frame_robot_1 = RDK.Item('UR3e_Base', robolink.ITEM_TYPE_FRAME)
    frame_robot_2 = RDK.Item('UR3e Base (2)', robolink.ITEM_TYPE_FRAME)

    #TARGETS
    home_1 = RDK.Item('HOME_R1', robolink.ITEM_TYPE_TARGET)
    home_2 = RDK.Item('HOME_R2', robolink.ITEM_TYPE_TARGET)
    safe_1 = RDK.Item('SAFE_R1', robolink.ITEM_TYPE_TARGET)
    safe_2 = RDK.Item('SAFE_R2', robolink.ITEM_TYPE_TARGET)

    # Asignar la herramienta al robot
    robot_1.setTool(tool_1)
    robot_2.setTool(tool_2)

    robot_1.setPoseFrame(frame_robot_1)
    robot_1.MoveJ(home_1)

    robot_2.setPoseFrame(frame_robot_2)
    robot_2.MoveJ(home_2)

    robot_1.setPoseFrame(frame_robot_1)
    robot_1.MoveJ(safe_1)

    robot_2.setPoseFrame(frame_robot_2)
    robot_2.MoveJ(safe_2)

def AvanzaSimpa():
    """
    Ejecuta un ciclo completo de la cinta transportadora:
    crea una nueva caja (si quedan), avanza la cinta 500mm y elimina
    las cajas que hayan salido del extremo.
    Decrementa los contadores de límite de cada sensor en cada llamada.
    """

    #----- Constantes -----
    NEW_REF_OBJECT_NAME = 'CAJA_REF'
    NEW_REF_OBJECT_NAME_2 = 'CAJA_REF_2'

    REFERENCE_FRAME = 'FrameCAJA'
    REFERENCE_FRAME_REF = 'FrameInitCaja'

    MECHANISM_NAME = 'CINTA_PRINCIPAL'
    MECHANISM_NAME_DOOR = 'Dispensa_CAJAS'

    PART_TRAVEL_MM = 500
    DOOR_TRAVEL_MM = 120

    #------- Program ------
    frame = RDK.Item(REFERENCE_FRAME, ITEM_TYPE_FRAME)
    frame_ref = RDK.Item(REFERENCE_FRAME_REF, ITEM_TYPE_FRAME)
    ref_obj = RDK.Item(NEW_REF_OBJECT_NAME, ITEM_TYPE_OBJECT)
    ref_obj_2 = RDK.Item(NEW_REF_OBJECT_NAME_2, ITEM_TYPE_OBJECT)


    door = RDK.Item(MECHANISM_NAME_DOOR,itemtype=robolink.ITEM_TYPE_ROBOT)
    mechanism = RDK.Item(MECHANISM_NAME,itemtype=ITEM_TYPE_ROBOT)

    #actualizar las variables de limite en cada avance
    p1 = int(RDK.getParam('TOTAL_PEDIDO_1'))
    p2 = int(RDK.getParam('TOTAL_PEDIDO_2'))

    LIMITE_TAPAS = int(RDK.getParam('LIMITE_TAPAS'))
    LIMITE_INSTRU = int(RDK.getParam('LIMITE_INSTRU'))
    LIMITE_BOLSAS = int(RDK.getParam('LIMITE_BOLSAS'))

    para = int(RDK.getParam('CICLOS_HASTA_PARAR'))

    if LIMITE_TAPAS > 0:
        LIMITE_TAPAS = LIMITE_TAPAS - 1

    if LIMITE_INSTRU > 0:
        LIMITE_INSTRU = LIMITE_INSTRU - 1

    if LIMITE_BOLSAS > 0:
        LIMITE_BOLSAS -= 1

    if para > 0:
        para = para - 1

    RDK.setParam('LIMITE_TAPAS', str(LIMITE_TAPAS))
    RDK.setParam('LIMITE_INSTRU', str(LIMITE_INSTRU))
    RDK.setParam('LIMITE_BOLSAS', str(LIMITE_BOLSAS))

    RDK.setParam('CICLOS_HASTA_PARAR', str(para))

    #CONTROL DE LA PARADA DE LA ESTACIoN
    if para <= 0:
        RDK.setParam('PARAR_ESTACION', '0')

    #Parar de generar pedidos cuando se hayan sacado todas las cajas
    if p1 == 0 and p2 == 0:
        RDK.setParam('PRODUCIR_CAJAS', '0')

    generar_nuevas_cajas = int(RDK.getParam('PRODUCIR_CAJAS'))

    #Mientras hayan cajas por crear, hacer copias
    if generar_nuevas_cajas == 1:

        seq = int(RDK.getParam('CONTADOR_CREADAS') or '0') + 1
        RDK.setParam('CONTADOR_CREADAS', str(seq))

        #INICIALIZAR PUERTA
        if door.Valid():
            door.setJoints([0])

        #CREAR COPIA DE CAJA
        RDK.Render(False)
        if p1 > 0:
            if frame.Valid() and  ref_obj.Valid():
                ref_obj.Copy()
                new_obj = RDK.Paste()
                new_obj.setVisible(False)
                new_obj.setName(f"CAJA_{seq:03d}")

                new_obj.setParent(frame_ref)
                RDK.Update()

                new_obj.setParentStatic(frame)
                new_obj.setVisible(True)

                #CAJA CREADA - SE RESTA DE LAS RESTANTES
                p1 = p1 - 1
                RDK.setParam('TOTAL_PEDIDO_1', str(p1))

        #igual para las cajas del segundo tipo
        elif p2 > 0:
            if frame.Valid() and  ref_obj.Valid():
                ref_obj_2.Copy()
                new_obj_2 = RDK.Paste()
                new_obj_2.setVisible(False)
                new_obj_2.setName(f"CAJA2_{seq:03d}")

                new_obj_2.setParent(frame_ref)
                RDK.Update()

                new_obj_2.setParentStatic(frame)
                new_obj_2.setVisible(True)

                p2 = p2 - 1
                RDK.setParam('TOTAL_PEDIDO_2', str(p2))

        RDK.Render(True)

    frame = frame.Childs()

    #Si la caja/objeto se encuentra fuera de la cinta se elimina
    for item in frame:
        try:
            if not item.Valid():
                continue
            if item.PoseAbs()[0,3] > 2100:
                item.Delete()
        except Exception:
            continue

    if generar_nuevas_cajas == 1:
        #ABRIR PUERTA
        if door.Valid():
            door.MoveJ(door.Joints() + DOOR_TRAVEL_MM)

    #Mover la cinta x distancia
    if mechanism.Valid():
        mechanism.MoveJ(mechanism.Joints() + PART_TRAVEL_MM)

    if generar_nuevas_cajas == 1:
        #CERRAR PUERTA
        if door.Valid():
            door.MoveJ(door.Joints() - DOOR_TRAVEL_MM)


# --- INICIO REAL DEL PROGRAMA PRINCIPAL ---
def programa_principal():
    Reset()

    # Esperar hasta recibir mensaje por MQTT
    while int(RDK.getParam('MQTT_ESTACION_ENCENDIDA')) == 0:
        time.sleep(0.1)

    #Hasta no recibir la señal mqtt no se puede actualizar las variables
    init()
    # Siempre debemos volver a encender los sensores
    RDK.RunProgram('DetectaSensor', False)

    if int(RDK.getParam('PARADA_EMERGENCIA')) == 1:
        return

    #caso que se pulse iniciar sin mandar nada
    if int(RDK.getParam('PEDIDO_2_INICIAL')) == 0 and int(RDK.getParam('PEDIDO_1_INICIAL')) == 0:
        return

    #Esperar a que la base de datos verifique el stock
    while int(RDK.getParam('STOCK_VERIFICADO')) == 0:
        if int(RDK.getParam('PARADA_EMERGENCIA')) == 1:
            break
        time.sleep(0.2)

    if int(RDK.getParam('PARADA_EMERGENCIA')) == 1:
        return

    #Mirar si se viene de una parada de emergencia
    es_reanudacion = int(RDK.getParam('ES_REANUDACION') or '0') == 1
    if not es_reanudacion:
        # COMPORTAMIENTO NORMAL: Forzar la primera caja
        AvanzaSimpa()
        time.sleep(0.2)

        if int(RDK.getParam('PARADA_EMERGENCIA')) == 0:
            contador_c = int(RDK.getParam('CONTADOR_C')) + 1
            RDK.setParam('CONTADOR_C', str(contador_c))
            RDK.setParam(f'NOMBRE_C_{contador_c:03d}', RDK.getParam('NOMBRE_CAJA_EN_C') or '')

            PEDIDO_1_INICIAL = int(RDK.getParam('PEDIDO_1_INICIAL'))
            RDK.setParam('R1_LIBRE', '0')   #indicamos que se esta realizando una accion en la estacion (parar cinta)

            if int(RDK.getParam('PEDIDO_2_INICIAL')) == 0 and int(RDK.getParam('PEDIDO_1_INICIAL')) == 0:
                return



            if contador_c > PEDIDO_1_INICIAL or int(RDK.getParam('PP_BOLSA_2')) == 1:
                RDK.RunProgram('ROBOT1_BOLSA2', False)
            else:
                RDK.RunProgram('ROBOT1_BOLSA1', False)
    else:
        # si viene de una emergencia, le damos medio segundo a los sensores
        time.sleep(0.5)


    # PROGRAMA GENERAL EN BUCLE HASTA QUE SE ACABEN LOS PEDIDOS
    while int(RDK.getParam('PARAR_ESTACION')) and int(RDK.getParam('PARADA_EMERGENCIA')) == 0:

        total_cajas = (int(RDK.getParam('PEDIDO_1_INICIAL')) + int(RDK.getParam('PEDIDO_2_INICIAL')))

        #Bucle para verificar que todos los procesos han acabado antes de avanzar la cinta de nuevo
        while int(RDK.getParam('R1_LIBRE')) == 0 or int(RDK.getParam('R2_LIBRE')) == 0 or int(RDK.getParam('INSTRU_LIBRE')) == 0:
            if int(RDK.getParam('PARADA_EMERGENCIA')) == 1:
                break
            time.sleep(0.1)

        #Lo coloco porque si en el bucle anterior hay emergencia, saltaba a lanzar la cinta automaticamente
        if int(RDK.getParam('PARADA_EMERGENCIA')) == 1:
            break

        #caso que se pulse iniciar sin mandar nada (por si acaso)
        if int(RDK.getParam('PEDIDO_2_INICIAL')) == 0 and int(RDK.getParam('PEDIDO_1_INICIAL')) == 0:
            return


        AvanzaSimpa()
        time.sleep(0.2)

    #COLOCAR BOLSAS
        if (int(RDK.getParam('LIMITE_BOLSAS')) != 0 and int(RDK.getParam('SenyalSensor_C')) == 1 and int(RDK.getParam('CONTADOR_C')) < total_cajas):

            contador_c = int(RDK.getParam('CONTADOR_C')) + 1
            RDK.setParam('CONTADOR_C', str(contador_c))
            RDK.setParam(f'NOMBRE_C_{contador_c:03d}', RDK.getParam('NOMBRE_CAJA_EN_C') or '')

            PEDIDO_1_INICIAL = int(RDK.getParam('PEDIDO_1_INICIAL'))

            #Se van contando las cajas ya montadas con las totales del tipo 1
            #También si el sensor detecta el tipo correcto, para asegurar fiabilidad
            if (contador_c > PEDIDO_1_INICIAL or int(RDK.getParam('PP_BOLSA_2')) == 1):
                es_tipo_2 = True
            else:
                es_tipo_2 = False

            RDK.setParam('R1_LIBRE', '0')
            if es_tipo_2:
                RDK.RunProgram('ROBOT1_BOLSA2', False)
            else:
                RDK.RunProgram('ROBOT1_BOLSA1', False)

    #COLOCAR INSTRUCCIONES
        if (int(RDK.getParam('LIMITE_INSTRU')) != 0 and int(RDK.getParam('SenyalSensor_I')) == 1 and int(RDK.getParam('CONTADOR_I')) < total_cajas):
            contador_i = int(RDK.getParam('CONTADOR_I')) + 1
            RDK.setParam('CONTADOR_I', str(contador_i))

            RDK.setParam('INSTRU_LIBRE', '0')
            RDK.RunProgram('PONER_INSTRU', False)

    #COLOCAR TAPA
        if (int(RDK.getParam('LIMITE_TAPAS')) != 0 and int(RDK.getParam('SenyalSensor_T')) == 1 and int(RDK.getParam('CONTADOR_T')) < total_cajas):
            contador_t = int(RDK.getParam('CONTADOR_T')) + 1
            RDK.setParam('CONTADOR_T', str(contador_t))
            RDK.setParam(f'NOMBRE_T_{contador_t:03d}', RDK.getParam('NOMBRE_CAJA_EN_T') or '')

            PEDIDO_1_INICIAL = int(RDK.getParam('PEDIDO_1_INICIAL'))

            if (contador_t > PEDIDO_1_INICIAL or int(RDK.getParam('TAPA_BOLSA_2')) == 1):
                es_tipo_2_t = True
            else:
                es_tipo_2_t = False

            RDK.setParam('R2_LIBRE', '0')
            if es_tipo_2_t:
                RDK.RunProgram('ROBOT2_TAPA2', False)
            else:
                RDK.RunProgram('ROBOT2_TAPA1', False)

        time.sleep(0.05)


    #Esperar a que los robots terminen
    while int(RDK.getParam('R1_LIBRE')) == 0 or int(RDK.getParam('R2_LIBRE')) == 0 or int(RDK.getParam('INSTRU_LIBRE')) == 0:
        if int(RDK.getParam('PARADA_EMERGENCIA')) == 1:
            break
        time.sleep(0.1)


def finalizar():
    if int(RDK.getParam('PARADA_EMERGENCIA')) == 0:
        #Devolver los robots a sus posiciones iniciales
        robot_1 = RDK.Item('r_UR3e_(COGIDA)', robolink.ITEM_TYPE_ROBOT)
        tool_1 = RDK.Item('VENTOSA-COG', robolink.ITEM_TYPE_TOOL)

        robot_2 = RDK.Item('r_UR3e_(TAPAS)', robolink.ITEM_TYPE_ROBOT)
        tool_2 = RDK.Item('VENTOSA-FIN', robolink.ITEM_TYPE_TOOL)

        #FRAMES
        frame_robot_1 = RDK.Item('UR3e_Base', robolink.ITEM_TYPE_FRAME)
        frame_robot_2 = RDK.Item('UR3e Base (2)', robolink.ITEM_TYPE_FRAME)

        #TARGETS
        home_1 = RDK.Item('HOME_R1', robolink.ITEM_TYPE_TARGET)
        home_2 = RDK.Item('HOME_R2', robolink.ITEM_TYPE_TARGET)
        safe_1 = RDK.Item('SAFE_R1', robolink.ITEM_TYPE_TARGET)
        safe_2 = RDK.Item('SAFE_R2', robolink.ITEM_TYPE_TARGET)

        robot_1.setTool(tool_1)
        robot_2.setTool(tool_2)

        robot_1.setPoseFrame(frame_robot_1)
        robot_1.MoveJ(home_1)

        robot_2.setPoseFrame(frame_robot_2)
        robot_2.MoveJ(home_2)

    #Asegurar que se para la estacion (por si se inicia sin pedidos)
    RDK.setParam('PARAR_ESTACION', '0')
    time.sleep(1)


if __name__ == "__main__":
    #Asegurar que estan en el valor deseado
    RDK.setParam('PARADA_EMERGENCIA', '0')
    RDK.setParam('ES_REANUDACION', '0')
    # Lanzamos los programas en segundo plano
    RDK.RunProgram('MqttListener', False)
    RDK.RunProgram('BASE_DATOS', False)

    # Bucle infinito del programa principal
    while 1:
        programa_principal()
        finalizar()

--- Python program MqttListener ---
import paho.mqtt.client as mqtt
from robodk import robolink
import json
import time
import ssl

RDK = robolink.Robolink()
"""
Stack Tecnológico: Python, Paho MQTT, ssl, json, RoboDK API.
Descripción: Script de comunicaciones asíncronas. Mantiene una conexión
viva vía WebSockets (WSS) con EMQX para recibir pedidos y órdenes de
emergencia desde un ESP32 o Dashboard, y notifica cuando la planta acaba.
"""
#Configuracion
broker="broker.emqx.io"
user="PR2_1_3"
passwd="public"

#Topics
base_topic="PR2_1_3/linea1"
topic_enviar=base_topic+"/python"
topic_recibir_esp=base_topic+"/esp"
topic_recibir_web=base_topic+"/web"

#Puertos
port_web=8084
port_esp=1883

def on_message_web(mqttc_web, obj, msg):
    """
    Callback disparado automáticamente cada vez que llega un mensaje al topic.
    Decodifica el JSON recibido. Si contiene cantidades de cajas, las guarda
    en RoboDK.
    """
    try:
        datos = json.loads(msg.payload.decode('utf-8'))

        #Recibir pedidos
        if "cajas_tipo_1" in datos:
            cantidad_1 = datos["cajas_tipo_1"]
            RDK.setParam('TOTAL_PEDIDO_1', str(cantidad_1))

        if "cajas_tipo_2" in datos:
            cantidad_2 = datos["cajas_tipo_2"]
            RDK.setParam('TOTAL_PEDIDO_2', str(cantidad_2))

    except json.JSONDecodeError:
        pass

def on_message_esp(mqttc_esp_cb, obj, msg):
    """
    Callback disparado automáticamente cada vez que llega un mensaje al topic.
    Decodifica el JSON recibido. Si es una orden de 'EMPIEZA' o 'EMERGENCIA', activa la estación
    o la detiene según corresponda.
    """
    try:
        #Convertir en json
        datos = json.loads(msg.payload.decode('utf-8'))

        #Encender la estacion
        if "tipo" in datos and datos["tipo"] == "EMPIEZA":
            if int(RDK.getParam('PARADA_EMERGENCIA') or '0') == 1:
                # Si había emergencia, la limpiamos y avisamos al Main
                RDK.setParam('PARADA_EMERGENCIA', '0')
                RDK.setParam('ES_REANUDACION', '1')
            else:
                # Si es un pedido nuevo limpio, generamos ID nuevo
                RDK.setParam('ES_REANUDACION', '0')
                id_pedido = f"PED_{int(time.time())}"
                RDK.setParam('NUMERO_PEDIDO', id_pedido)

            RDK.setParam('MQTT_ESTACION_ENCENDIDA', '1')
            mqttc_esp.publish(topic_enviar, json.dumps({"tipo": "PLANTA_ACTIVA"}))

        #Boton de emergencia
        if "tipo" in datos and datos["tipo"] == "EMERGENCIA":
            RDK.setParam('PARADA_EMERGENCIA', '1')

            mensaje = json.dumps({"tipo": "PLANTA_INACTIVA"})
            mqttc_esp.publish(topic_enviar, mensaje)

    except json.JSONDecodeError:
        pass

def on_connect_esp(client, userdata, flags, reason_code, properties):
    """
    Callback disparado automáticamente cuando se establece la conexión con el broker.
    Se suscribe inmediatamente al topic de escucha de la ESP (topic_enviar).
    """
    client.subscribe(topic_recibir_esp, 0)

def on_connect_web(client, userdata, flags, reason_code, properties):
    """
    Callback disparado automáticamente cuando se establece la conexión con el broker.
    Se suscribe inmediatamente al topic de escucha de la web (topic_enviar) (para recibir los pedidos).
    """
    client.subscribe(topic_recibir_web, 0)

#Cliente web
mqttc_web = mqtt.Client(
    mqtt.CallbackAPIVersion.VERSION2,
    transport="websockets",
    protocol=mqtt.MQTTv311
)

mqttc_web.on_connect = on_connect_web
mqttc_web.on_message = on_message_web
mqttc_web.username_pw_set(username=user, password=passwd)
mqttc_web.ws_set_options(path="/mqtt")
mqttc_web.tls_set()
mqttc_web.connect(broker, port_web, 60)
mqttc_web.loop_start()

#Cliente ESP
mqttc_esp = mqtt.Client(mqtt.CallbackAPIVersion.VERSION2)
mqttc_esp.on_connect = on_connect_esp
mqttc_esp.on_message = on_message_esp
mqttc_esp.username_pw_set(username=user, password=passwd)
mqttc_esp.connect(broker, port_esp, 60)
mqttc_esp.loop_start()


#Enviar mensaje que la estacion ya ha acabado
estado_actual = -1
estado_anterior = 0
while True:
    try:
        estado_actual = int(RDK.getParam('PARAR_ESTACION'))
    except:
        estado_actual = 0

    if estado_actual == 0 and estado_anterior == 1:
        mensaje = json.dumps({"tipo": "PLANTA_INACTIVA"})
        mqttc_esp.publish(topic_enviar, mensaje)
        time.sleep(0.3)   # dar margen para que el publish salga antes de desconectar

    estado_anterior = estado_actual
    time.sleep(0.5)

--- Python program BASE_DATOS ---
import time
import psycopg
from robodk import robolink
from datetime import datetime

RDK = robolink.Robolink()

""""
Stack Tecnológico: Python, Paho MQTT, ssl, json, RoboDK API, pgAdmin4.
Descripción: Encargado de conectarse a la base de datos LOCAL del sistema.
Revisa continuamente los movimientos realizados en la simulación para
registrar/actualizar los campos de la tabla Cajas de la base de datos.
También revisa antes de empezar a producir el stock actual.
"""

# Configuración BD
DB_CONFIG = {
    "dbname":   "gdi",
    "user":     "postgres",
    "password": "postgres",
    "host":     "localhost",
    "port":     "5432"
}

# Códigos de componentes
COD_CAJA_VACIA = "C001"
COD_BOLSA_A    = "C002"
COD_BOLSA_B    = "C003"
COD_TAPA       = "C004"
COD_MANUAL     = "C005"

# Códigos de tipo de caja
TIPO_AMARILLA = "TC01"
TIPO_ROJA     = "TC02"


# FUNCIONES DE BASE DE DATOS
def get_connection():
    return psycopg.connect(**DB_CONFIG)


def db_check_stock_preciso(codigo, cantidad_necesaria):
    """Comprueba que el stock actual cubre exactamente la cantidad del pedido."""
    conn = cur = None
    try:
        conn = get_connection()
        cur  = conn.cursor()
        cur.execute("SELECT Stock_Actual FROM Almacen WHERE Codigo = %s", (codigo,))
        fila = cur.fetchone()

        if fila:
            stock_actual = fila[0]
            if stock_actual >= cantidad_necesaria:
                return True
            else:
                return False
        return False

    except Exception as e:
        return False

    finally:
        if cur:  cur.close()
        if conn: conn.close()


def db_registrar_pedido(num_localizador):
    """Crea el registro del pedido en Pedido si no existe."""
    conn = cur = None
    try:
        conn = get_connection()
        cur  = conn.cursor()
        sql  = """
            INSERT INTO Pedido (Numero_Localizador, Fecha_Pedido, DNI_CIF)
            VALUES (%s, CURRENT_DATE,
                (SELECT DNI_CIF FROM Cliente LIMIT 1))
            ON CONFLICT (Numero_Localizador) DO NOTHING
        """
        cur.execute(sql, (num_localizador,))
        conn.commit()

    except Exception as e:
        if conn: conn.rollback()

    finally:
        if cur:  cur.close()
        if conn: conn.close()


def db_registrar_caja(cod_fisico, tipo_num, num_localizador):
    """
    Inserta la caja en la tabla Caja cuando pasa por el sensor C.
    cod_fisico es el ID único (ej: LEGO_PED_001_001).
    tipo_num: 1 = Amarilla, 2 = Roja.
    """
    cod_tipo    = TIPO_AMARILLA if tipo_num == 1 else TIPO_ROJA
    nombre_tipo = "Caja Amarilla T1" if tipo_num == 1 else "Caja Roja T2"
    conn = cur  = None
    try:
        conn = get_connection()
        cur  = conn.cursor()
        sql  = """
            INSERT INTO Caja (cod, tipo, acabada, numero_localizador, codigo_tipo)
            VALUES (%s, %s, FALSE, %s, %s)
        """
        cur.execute(sql, (cod_fisico, nombre_tipo, num_localizador, cod_tipo))
        conn.commit()

    except Exception as e:
        if conn: conn.rollback()

    finally:
        if cur:  cur.close()
        if conn: conn.close()


def db_finalizar_caja(cod_fisico, tiempo_segundos=None):
    """
    Marca Acabada=TRUE y guarda el tiempo de producción cuando la caja
    pasa por el sensor T (tapa colocada).
    """
    conn = cur = None
    try:
        conn = get_connection()
        cur  = conn.cursor()
        sql  = "UPDATE Caja SET acabada = TRUE, tiempo_produccion = %s WHERE cod = %s"
        cur.execute(sql, (round(tiempo_segundos, 1) if tiempo_segundos else None, cod_fisico))
        conn.commit()

    except Exception as e:
        if conn: conn.rollback()

    finally:
        if cur:  cur.close()
        if conn: conn.close()


def db_descontar_stock(lista_componentes):
    """Resta 1 unidad por cada componente de la lista."""
    conn = cur = None
    try:
        conn = get_connection()
        cur  = conn.cursor()
        cur.executemany(
            "UPDATE Almacen SET Stock_Actual = Stock_Actual - 1 WHERE Codigo = %s",
            [(c,) for c in lista_componentes]
        )
        conn.commit()

    except Exception as e:
        if conn: conn.rollback()

    finally:
        if cur:  cur.close()
        if conn: conn.close()


def _leer_param(nombre, default=""):
    try:
        val = RDK.getParam(nombre)
        return val if val else default
    except Exception:
        return default


# LÓGICA PRINCIPAL
def run():
    while True:

        #Esperar arranque
        while int(_leer_param('MQTT_ESTACION_ENCENDIDA', '0')) == 0:
            time.sleep(0.5)

        # Esperar a que init() termine de escribir los parámetros
        time.sleep(1.0)

        #Leer datos del pedido
        num_localizador = _leer_param('NUMERO_PEDIDO', 'DESCONOCIDO')
        p1 = int(_leer_param('PEDIDO_1_INICIAL', '0'))
        p2 = int(_leer_param('PEDIDO_2_INICIAL', '0'))
        total_t1 = p1
        total_cajas = p1 + p2

        if total_cajas == 0:
            continue
        else:
            # Reanudación o pedido nuevo
            es_reanudacion = int(_leer_param('ES_REANUDACION', '0')) == 1

            mapa_cajas    = {}
            tiempos_inicio = {}

            if es_reanudacion:
                # Restaurar desde los contadores que quedaron en RoboDK
                prev_c = int(_leer_param('CONTADOR_C', '0'))
                prev_t = int(_leer_param('CONTADOR_T', '0'))
                prev_i = int(_leer_param('CONTADOR_I', '0'))

                # Reconstruir mapa para cajas que pasaron C pero no T
                # Usamos MAPA_CAJA_{i} que Base_datos guarda en cada evento C
                for i in range(prev_t + 1, prev_c + 1):
                    nombre_rdk = _leer_param(f'MAPA_CAJA_{i:03d}', '')
                    if nombre_rdk:
                        id_fisico = f"LEGO_{num_localizador}_{i:03d}"
                        mapa_cajas[nombre_rdk] = id_fisico
                        tiempos_inicio[id_fisico] = time.time()

                RDK.setParam('STOCK_VERIFICADO', '1')

            else:
                prev_c = 0
                prev_t = 0
                prev_i = 0

                # Comprobar stock
                comprobaciones = [
                    (COD_CAJA_VACIA, total_cajas),
                    (COD_BOLSA_A,    p1),
                    (COD_BOLSA_B,    p2),
                    (COD_TAPA,       total_cajas),
                    (COD_MANUAL,     total_cajas),
                ]
                stock_ok = all(
                    db_check_stock_preciso(cod, qty)
                    for cod, qty in comprobaciones if qty > 0
                )

                if not stock_ok:
                    RDK.ShowMessage(
                        f"PRODUCCIÓN BLOQUEADA: Stock insuficiente para el pedido "
                        f"{num_localizador}. Reponga el almacén y envíe un nuevo pedido.",
                        False
                    )
                    RDK.setParam('PARADA_EMERGENCIA', '1')
                    while int(_leer_param('MQTT_ESTACION_ENCENDIDA', '0')) == 1:
                        time.sleep(1.0)
                    continue

                # Registrar el pedido en BD y autorizar arranque
                db_registrar_pedido(num_localizador)
                RDK.setParam('STOCK_VERIFICADO', '1')

            #Bucle de vigilancia
            while (int(_leer_param('PARAR_ESTACION', '1')) == 1 and int(_leer_param('MQTT_ESTACION_ENCENDIDA','0')) == 1):

                #  Sensor C: nueva caja entra a producción
                curr_c = int(_leer_param('CONTADOR_C', '0'))
                if curr_c > prev_c:
                    for i in range(prev_c + 1, curr_c + 1):
                        #identificar la caja
                        tipo_num   = 1 if i <= total_t1 else 2
                        nombre_rdk = f"CAJA_{i:03d}" if tipo_num == 1 else f"CAJA2_{i:03d}"

                        id_fisico  = f"LEGO_{num_localizador}_{i:03d}"
                        cod_bolsa  = COD_BOLSA_A if tipo_num == 1 else COD_BOLSA_B

                        mapa_cajas[nombre_rdk]      = id_fisico
                        tiempos_inicio[id_fisico]   = time.time()
                        RDK.setParam(f'MAPA_CAJA_{i:03d}', nombre_rdk)

                        db_registrar_caja(id_fisico, tipo_num, num_localizador)
                        db_descontar_stock([COD_CAJA_VACIA, cod_bolsa])
                    prev_c = curr_c

                # Sensor T: tapa colocada -> caja acabada
                curr_t = int(_leer_param('CONTADOR_T', '0'))
                if curr_t > prev_t:
                    for i in range(prev_t + 1, curr_t + 1):

                        tipo_num_t = 1 if i <= total_t1 else 2
                        nombre_matematico = f"CAJA_{i:03d}" if tipo_num_t == 1 else f"CAJA2_{i:03d}"

                        id_fisico = mapa_cajas.get(nombre_matematico)

                        if id_fisico:
                            db_descontar_stock([COD_TAPA])
                            db_descontar_stock([COD_MANUAL])
                            tiempo_total = time.time() - tiempos_inicio.get(id_fisico, time.time())
                            db_finalizar_caja(id_fisico, tiempo_total)
                        else:
                            continue
                    prev_t = curr_t

                # Salida de emergencia
                if int(_leer_param('PARADA_EMERGENCIA', '0')) == 1:
                    print(f"[DB] Emergencia detectada. Suspendiendo pedido {num_localizador}.")
                    break

                time.sleep(0.5)

            # Drenaje: procesar cajas en tránsito
            tiempo_espera = 0
            while prev_t < prev_c and tiempo_espera < 60:

                curr_t = int(_leer_param('CONTADOR_T', '0'))
                if curr_t > prev_t:
                    for i in range(prev_t + 1, curr_t + 1):
                        tipo_num_t = 1 if i <= total_t1 else 2
                        nombre_matematico = f"CAJA_{i:03d}" if tipo_num_t == 1 else f"CAJA2_{i:03d}"

                        id_fisico = mapa_cajas.get(nombre_matematico)

                        if id_fisico:
                            db_descontar_stock([COD_TAPA])
                            db_descontar_stock([COD_MANUAL])
                            tiempo_total = time.time() - tiempos_inicio.get(id_fisico, time.time())
                            db_finalizar_caja(id_fisico, tiempo_total)
                    prev_t = curr_t

                if int(_leer_param('PARADA_EMERGENCIA', '0')) == 1:
                    break

                time.sleep(0.5)
                tiempo_espera += 0.5


if __name__ == "__main__":
    run()
